TYPE ST_DebugSensors_TransferCCEmulation :
STRUCT
	EnableSensorDebug	: BOOL; 					// Overwrite sensor values with debug sensor values
	HW_Inputs			: ST_HW_InputsTransferCC;	// Debug sensors
END_STRUCT
END_TYPE

(* stored: Version 1.1.0.1, ProductVersion 3.1.4024.9
   DUT ST_DebugSensors_TransferCCEmulation: Id {e80ae0af-6506-44e4-bbef-6b4903da6383} *)
